TYPE ST_RejectReason :
STRUCT
	Reason	:STRING;
END_STRUCT
END_TYPE

(* stored: Version 1.1.0.1, ProductVersion 3.1.4024.13
   DUT ST_RejectReason: Id {fe597c8e-b5f0-44f2-b1e3-037ccc9c2f0b} *)
